TYPE ST_ConveyorInputs :
STRUCT
	bConveyorIsMoving	:BOOL;
	bConveyorStopped	:BOOL;
	bPartDetected		:BOOL;
	bPartAvailable2Move	:BOOL;
	bRobInSpace			:BOOL;
END_STRUCT
END_TYPE

(* stored: Version 1.1.0.1, ProductVersion 3.1.4024.16
   DUT ST_ConveyorInputs: Id {e06003f2-3484-4b36-9c3d-8d77d369ce5d} *)
